{attribute 'qualified_only'}
TYPE E_AxisMode :
(
	INIT,
	ENABLE,
	JOG,
	POSITIONING,
	STOP,
	RESET,
	ERROR
);
END_TYPE

(* stored: Version 1.1.0.1, ProductVersion 3.1.4022.10
   DUT E_AxisMode: Id {14616915-b245-4e9a-b075-84ec09ec9f85} *)
